// TIA Portal V20 export
TYPE "typeSequenceControlNodeJobInterface"
// stored: Namespace Unit1.Em6
   STRUCT
      loadJob2 : "LER_typeJobInterface";
      inspectionJob3 : "LER_typeJobInterface";
      unloadJob4 : "LER_typeJobInterface";
   END_STRUCT;
END_TYPE
